// TIA Portal V17 export
// export: Created 2025-04-16T11:30:16.1752927Z, ExportSetting WithDefaults, DisplayName Totally Integrated Automation Portal, DisplayVersion V17, DisplayName TIA Portal Openness, DisplayVersion V17, DisplayName TIA Portal Version Control Interface, DisplayVersion V17, DisplayName STEP 7 Professional, DisplayVersion V17, DisplayName STEP 7 Safety, DisplayVersion V17, DisplayName WinCC Advanced, DisplayVersion V17
DATA_BLOCK "io"   // DB1
{ S7_Optimized_Access := 'TRUE' }
VERSION : 0.1
// stored: AutoNumber true, DBAccessibleFromOPCUA true, IsOnlyStoredInLoadMemory false, IsRetainMemResEnabled false, IsWriteProtectedInAS false, MemoryReserve 100
   VAR
      i : Struct
         a0 : Bool;
         a1 : Bool;
         b0 : Bool;
         b1 : Bool;
         c0 : Bool;
         c1 : Bool;
         d0 : Bool;
         d1 : Bool;
         mode : Bool;
         start : Bool;
         stop : Bool;
         pres : Bool;
         ma : Bool;
         mb : Bool;
         mc : Bool;
         md : Bool;
      END_STRUCT;
      "m" : Struct
         alap_start : Bool;
         alap : Bool;
         mode : Bool;
         step_no : Int;
         betanit_mode : Bool;
         mem : Struct
            ma1 : Bool;
            ma2 : Bool;
            ma3 : Bool;
            ma4 : Bool;
            ma5 : Bool;
            ma6 : Bool;
            ma7 : Bool;
            ma8 : Bool;
            mb1 : Bool;
            mb2 : Bool;
            mb3 : Bool;
            mb4 : Bool;
            mb5 : Bool;
            mb6 : Bool;
            mb7 : Bool;
            mb8 : Bool;
            mc1 : Bool;
            mc2 : Bool;
            mc3 : Bool;
            mc4 : Bool;
            mc5 : Bool;
            mc6 : Bool;
            mc7 : Bool;
            mc8 : Bool;
            md1 : Bool;
            md2 : Bool;
            md3 : Bool;
            md4 : Bool;
            md5 : Bool;
            md6 : Bool;
            md7 : Bool;
            md8 : Bool;
         END_STRUCT;
      END_STRUCT;
      o : Struct
         auto : Bool;
         run : Bool;
         "20" : Bool;
         "21" : Bool;
         "22" : Bool;
         pres : Bool;
         man : Bool;
         err : Bool;
         ma : Bool;
         mb : Bool;
         mc : Bool;
         md : Bool;
      END_STRUCT;
   END_VAR
BEGIN
END_DATA_BLOCK
